(* PLC project Unnamed, Unknown Unnamed 1 *)
(* stored: creationDateTime 2026-01-25T18:15:32, modificationDateTime 2026-01-25T18:15:32 *)

PROGRAM main
  VAR
    Temp AT %MW0 : INT := 260;  (* Simulated temperature in tenths of °C *)
    FanCmd AT %QX0.0 : BOOL := FALSE;  (* Cooling fan ON/OFF output *)
  END_VAR
  VAR
    HighT : INT := 230;  (* High threshold = 23.0 °C *)
    LowT : INT := 210;  (* Low threshold = 21.0 °C *)
  END_VAR

            (* If temp is high enough, turn fan ON *)
IF Temp >= HighT THEN
    FanCmd := TRUE;

(* If tempe is low enough, turn fan OFF *)
ELSIF Temp <= LowT THEN
    FanCmd := FALSE;
END_IF;
          
END_PROGRAM

CONFIGURATION Config0
  RESOURCE Res0 ON PLC
    TASK task0(INTERVAL := T#20ms, PRIORITY := 1);
    PROGRAM instance0 WITH task0 : main;
  END_RESOURCE
END_CONFIGURATION
